PROGRAM MAIN
VAR
    fbGetmA: FB_AnalogInput;
    fmA: LREAL;
    {attribute 'TcLinkTo' := 'TIID^Device 1 (EtherCAT)^Term 1 (EK1200)^Term 2 (EL3052)^AI Standard Channel 1^Value'}
    rawInputmA AT %I*: INT;


    {attribute 'pytmc' := 'pv: XBD:N2:MAX_MASS'}
    maxMass: LREAL;
    {attribute 'pytmc' := 'pv: XBD:N2:MIN_MASS'}
    minMass: LREAL;
    {attribute 'pytmc' := 'pv: XBD:N2:CURRENT_MASS'}
    fMassofGas: LREAL;
    {attribute 'pytmc' := 'pv: XBD:N2:MAINTENANCE_MODE'}
    bMaintenanceMode : BOOL := FALSE;

    {attribute 'pytmc' := 'pv: XBD:N2:LOW_LEVEL'}
    fMassLowLevl : LREAL := maxMass / 2;
    bMassIsLow : BOOL := FALSE;

    fbValveTimer : TON;
    fbCloseValveTimer : TOF;

    fbValveRelay : FB_VALVE_RELAY;

    bInit : BOOL := TRUE;
    iState : INT  := 0;

END_VAR

IF bInit THEN
    maxMass := 500;
    minMass := 0;
    bInit := FALSE;
    fbValveTimer.PT := T#1m; // SET FOR 1 MIN FOR TESTING
    fbCloseValveTimer.PT := T#1s; // TIME VALVE SHOULD REMAIN OPEN
END_IF

fbValveTimer(IN:=TRUE); // RUN TIMER
fbCloseValveTimer(IN:= FALSE); // RUN OFF TIMER

fbValveRelay();

fbGetmA(
    iRaw := rawInputmA,
    iTermBits := 12,
    fTermMax := 20,
    fTermMin := 4,
    fReal => fmA
);

fMassofGas := (fmA - 4.0) / 16.0 * maxMass + minMass;

CASE iState OF
    0: // INIT
    fbValveTimer(IN:=FALSE); //RESTART TIMER
    IF NOT bMaintenanceMode THEN
        iState := 2;
    END_IF

    1: // MAINTINANCE MODE
    IF NOT bMaintenanceMode THEN
        iState := 0;
        fbCloseValveTimer(IN:= TRUE); // ACTUATE VALE AFTER EXIT MAINTINACE MODE
    END_IF

    2: // OP MODE

    IF fMassofGas < fMassLowLevl THEN bMassIsLow := TRUE; ELSE bMassIsLow := FALSE; END_IF;

    //rawOutputRelayChan1 := NOT bMassIsLow; // OPEN IF MASS IS NOT LOW and CLOSE IF MASS IS LOW

    IF bMassIsLow AND fbCloseValveTimer.Q THEN
        //rawOutputRelayChan1 := fbCloseValveTimer.Q;
    END_IF

    IF NOT bMassIsLow AND fbCloseValveTimer.Q THEN
        //rawOutputRelayChan1 := NOT fbCloseValveTimer.Q;
    END_IF

    // ACTUAVE VALVE EVERY 24 HOURS
    IF fbValveTimer.Q THEN
        fbValveTimer(IN:=FALSE); //RESTART TIMER
        fbCloseValveTimer(IN:= TRUE); // RUN OFF TIMER
    END_IF

    IF bMaintenanceMode THEN
        iState := 1;
        //rawOutputRelayChan1 := FALSE; // CLOSE VALVE WHEN ENTERING MAINTINANCE MODE
    END_IF
END_CASE

END_PROGRAM

(* stored: Version 1.1.0.1, ProductVersion 3.1.4024.11
   POU MAIN: Id {33620bff-f8ff-418a-9b35-0303bd8eb7b6}, SpecialFunc None *)
